Staubli VAL3: onF3Event.pgx

program onF3Event()
  local string l_sItem
  local string l_sPage
begin
  // look if the bButton is enable
  if bButton[2]
    //
    l_sPage="Disk://instruction/inputOutput/page_inOut"
    call loadPage(l_sPage,l_sItem)
    //
    logMsg("[KERNEL] INTERFACE:PAGE Home Page")
  endIf
end
